{attribute 'linkalways'} 
{attribute 'no_explicit_call' := 'This FB is a CLASS and must be accessed using methods or properties'}
{attribute 'enable_dynamic_creation'}
FUNCTION_BLOCK FINAL LT_UDINT EXTENDS Node
VAR
	in1 : _UDINT(0);
	in2 : _UDINT(0);
	out : _BOOL(FALSE);
END_VAR

METHOD PUBLIC Clone : I_Node
VAR
	pNode : POINTER TO LT_UDINT;
END_VAR
pNode := __NEW(LT_UDINT);
Clone := pNode^;
END_METHOD

METHOD FB_init : BOOL
VAR_INPUT
	bInitRetains : BOOL; // if TRUE, the retain variables are initialized (warm start / cold start)
	bInCopyCode : BOOL;  // if TRUE, the instance afterwards gets moved into the copy code (online change)
END_VAR
AddInput('in1',THIS^.in1);
AddInput('in2',THIS^.in2);
AddOutput('out', THIS^.out);
END_METHOD

METHOD PROTECTED OnExecute
VAR
END_VAR
out.Value := in1.Value < in2.Value;
END_METHOD

END_FUNCTION_BLOCK

(* stored: Version 1.1.0.1, ProductVersion 3.1.4024.15
   POU LT_UDINT: Id {a714ff13-b1c2-4788-826a-43bbf7e81e52}, SpecialFunc None
   Folder Constructor: Id {1c3f03ec-0e93-4686-829c-d32a59088677}
   Method Clone: Id {884b2cdd-e3c5-478f-bea8-30c9636eb720}
   Method FB_init: Id {07258c87-5549-4a93-b182-766f53d3170a}
   Method OnExecute: Id {a71c3d6c-4989-482e-b9ec-cccc1a1b235b} *)
